// TIA Portal V17 export
// export: Created 2025-06-25T13:13:24.7047341Z, ExportSetting WithDefaults, DisplayName Totally Integrated Automation Portal, DisplayVersion V17 Update 8, DisplayName TIA Portal Openness, DisplayVersion V17 Update 8, DisplayName TIA Portal Version Control Interface, DisplayVersion V17, DisplayName STEP 7 Professional, DisplayVersion V17 Update 8, DisplayName STEP 7 Safety, DisplayVersion V17 Update 6, DisplayName WinCC Advanced, DisplayVersion V17 Update 8
DATA_BLOCK "DB_Calc"   // DB45
{ S7_Optimized_Access := 'FALSE' }
AUTHOR : Heaten
VERSION : 0.1
// stored: AutoNumber true, DBAccessibleFromOPCUA true, DBAccessibleFromWebserver true, IsOnlyStoredInLoadMemory false, IsWriteProtectedInAS false
   VAR RETAIN
      Compressor : Struct
         CrankcaseSaturationTemperature : "stCalcValue";   // C
         CrankcaseSuperheat { S7_SetPoint := 'True'} : "stCalcValue";
         VolumetricEfficiency { S7_SetPoint := 'True'} : "stCalcValue";   // %
         IsentropicEfficiency { S7_SetPoint := 'True'} : "stCalcValue";   // %
         Massflow { S7_SetPoint := 'True'} : "stCalcValue";   // Refrigerant massflow (kg/h)
      END_STRUCT;
      HeatSink : Struct
         DeltaT : "stCalcValue";   // C
         Pinch { S7_SetPoint := 'True'} : "stCalcValue";   // C
         HeatRate { S7_SetPoint := 'True'} : "stCalcValue";   // kW
         DeltaP { S7_SetPoint := 'True'} : "stCalcValue";   // kPa
         Massflow { S7_SetPoint := 'True'} : "stCalcValue";   // Cooling media massflow (t/h)
      END_STRUCT;
      HeatSource : Struct
         DeltaT : "stCalcValue";   // C
         Pinch { S7_SetPoint := 'True'} : "stCalcValue";   // C
         HeatRate { S7_SetPoint := 'True'} : "stCalcValue";   // kW
         DeltaP { S7_SetPoint := 'True'} : "stCalcValue";   // kPa
         TemperatureRateOfChange { S7_SetPoint := 'True'} : "stCalcValue";   // C/s
         Massflow { S7_SetPoint := 'True'} : "stCalcValue";   // Heating media massflow (t/h)
      END_STRUCT;
      HighPressPart : Struct
         CompressorSaturationTemperature : "stCalcValue";
         CompressorSuperheat : "stCalcValue";   // C
         CondenserSaturationTemperature : "stCalcValue";   // C
         CondenserSubcooling : "stCalcValue";   // C
         ExpansionValveSubcooling : "stCalcValue";   // C
         CondenserDeltaP : "stCalcValue";   // kPa
      END_STRUCT;
      LowPressPart : Struct
         EvaporatorSuperheat : "stCalcValue";   // C
         CompressorSuperheat { S7_SetPoint := 'True'} : "stCalcValue";   // C
         EvaporatorSaturationTemperature { S7_SetPoint := 'True'} : "stCalcValue";   // C
         CompressorSaturationTemperature { S7_SetPoint := 'True'} : "stCalcValue";   // C
      END_STRUCT;
      System : Struct
         Quality : "stCalcValue";   // 1
         COP { S7_SetPoint := 'True'} : "stCalcValue";   // 1
         ElectricalPower { S7_SetPoint := 'True'} : "stCalcValue";   // kW
         TemperatureLift { S7_SetPoint := 'True'} : "stCalcValue";   // C
         MotorEfficiency { S7_SetPoint := 'True'} : "stCalcValue";   // Instantaneous efficiency (%)
         FMEP { S7_SetPoint := 'True'} : "stCalcValue";   // kPa
      END_STRUCT;
      Auxiliary : Struct
         ShaftSealDeltaT : "stCalcValue";   // C
         CPCDeltaP { S7_SetPoint := 'True'} : "stCalcValue";
      END_STRUCT;
      Misc : Struct
         EvaporatorDischargePressureMean { S7_SetPoint := 'True'} : "stCalcValue";   // Average of Evaporator A & B discharge pressures
         EvaporatorDischargeTemperatureMin { S7_SetPoint := 'True'} : "stCalcValue";   // Smaller of Evaporator A & B discharge temperatures
         EvaporatorDischargeTemperatureMean { S7_SetPoint := 'True'} : "stCalcValue";   // Average of Evaporator A & B discharge temperatures
         OilFilterDeltaP { S7_SetPoint := 'True'} : "stCalcValue";   // kPa
      END_STRUCT;
   END_VAR
BEGIN
   HeatSink.DeltaP.fMin := 0.0;
   HeatSink.DeltaP.fMax := 1000.0;
   HeatSink.DeltaP.bCheckLimits := TRUE;
   HeatSource.DeltaP.fMax := 4000.0;
   HeatSource.DeltaP.bCheckLimits := true;
END_DATA_BLOCK
